(* CODESYS project shelf.library
   Title: Shelf
   Company: Stefan Lehmann
   Version: 0.0.1
   Placeholder: Shelf

Project tree, tasks and I/O mapping:
  libraries: Tc2_System, * (Beckhoff Automation GmbH); Tc2_Utilities, * (Beckhoff Automation GmbH); Tc3_Module, * (Beckhoff Automation GmbH)
  classes/
    function block FifoBuffer [ST]: A_Add, A_Get, A_Remove, A_Reset
    function block Part [ST]: FB_init, id
    function block Shelf [ST]: FB_init, getNextFreeSpace, getNextOccupiedSpace, getShelfSpaceByPartId, m, n, storeNextPart, unloadNextPart, unloadPartById
    function block ShelfElement [ST]: column, isOccupied, part, row, store, unload
  interfaces/
    interface IPart: id
    interface IShelf: getNextFreeSpace, getNextOccupiedSpace, getShelfSpaceByPartId, m, n, storeNextPart, unloadNextPart, unloadPartById
    interface IShelfElement: column, isOccupied, part, row, store, unload
  ClassDiagram
  program main [ST]
*)

// classes/FifoBuffer
FUNCTION_BLOCK FifoBuffer
VAR_INPUT
	bOverwrite	: BOOL;
	in 			: IShelfElement;
END_VAR
VAR_OUTPUT
	bOk			: BOOL;
	nCount		: UDINT;
	nLoad		: UDINT;
	out			: IShelfElement;
END_VAR
VAR
	arrBuffer 	: ARRAY[0..MAX_BUFFER_SIZE] OF BYTE; (* Buffer memory used by FB_MemRingBuffer function block *)
	fbBuffer	: FB_MemRingBuffer;
END_VAR
VAR CONSTANT
	MAX_BUFFER_SIZE : UDINT := 1000;
END_VAR

;

ACTION A_Add:
fbBuffer.A_AddTail( pWrite:= ADR( in ),
					cbWrite:= SIZEOF( in ),
					pBuffer:= ADR( arrBuffer ),
					cbBuffer:= SIZEOF( arrBuffer ),
					bOk=> bOk,
					nCount => nCount );


IF NOT bOk THEN (* overflow ? *)
	IF bOverwrite THEN
		fbBuffer.A_RemoveHead(); (* remove one oldest entry *)

		fbBuffer.A_AddTail( bOk => bOk, nCount => nCount );
	END_IF
END_IF



nLoad := (fbBuffer.cbSize * 100) / MAX_BUFFER_SIZE;
END_ACTION

ACTION A_Get:
fbBuffer.A_GetHead( pRead:= ADR( out ),
					cbRead:= SIZEOF( out ),
					pBuffer:= ADR( arrBuffer ),
					cbBuffer:= SIZEOF( arrBuffer ),
					bOk=> bOk,
					nCount => nCount );

nLoad := (fbBuffer.cbSize * 100) / MAX_BUFFER_SIZE;
END_ACTION

ACTION A_Remove:
fbBuffer.A_RemoveHead( 	pRead:= ADR( out ),
						cbRead:= SIZEOF( out ),
						pBuffer:= ADR( arrBuffer ),
						cbBuffer:= SIZEOF( arrBuffer ),
						bOk=> bOk,
						nCount => nCount );

nLoad := (fbBuffer.cbSize * 100) / MAX_BUFFER_SIZE;
END_ACTION

ACTION A_Reset:
MEMSET( ADR( arrBuffer ), 0, SIZEOF( arrBuffer ) ); (* reset (optional) internal buffer *)

fbBuffer.A_Reset( 	bOk=> bOk,
					nCount => nCount );

nLoad := (fbBuffer.cbSize * 100) / MAX_BUFFER_SIZE;
END_ACTION

END_FUNCTION_BLOCK

// interfaces/IShelfElement
INTERFACE IShelfElement EXTENDS __System.IQueryInterface

PROPERTY column : UINT
GET
END_GET
SET
END_SET
END_PROPERTY

PROPERTY isOccupied : BOOL
GET
END_GET
END_PROPERTY

PROPERTY part : IPart
GET
END_GET
END_PROPERTY

PROPERTY row : UINT
GET
END_GET
SET
END_SET
END_PROPERTY

METHOD store : BOOL
VAR_INPUT
	part: IPart;
END_VAR
END_METHOD

METHOD unload : IPart
VAR_INPUT
END_VAR
END_METHOD

END_INTERFACE

// classes/Part
FUNCTION_BLOCK Part IMPLEMENTS IPart
VAR_INPUT
END_VAR
VAR_OUTPUT
END_VAR
VAR
	_id: STRING(23);
END_VAR

//FB_Init is always available implicitly and it is used primarily for initialization.
//The return value is not evaluated. For a specific influence, you can also declare the
//methods explicitly and provide additional code there with the standard initialization
//code. You can evaluate the return value.
METHOD FB_Init: BOOL
VAR_INPUT
    bInitRetains: BOOL; // TRUE: the retain variables are initialized (reset warm / reset cold)
    bInCopyCode: BOOL;  // TRUE: the instance will be copied to the copy code afterward (online change)
	id: String(23);   
END_VAR
THIS^._id := id;
END_METHOD

{warning 'Eigenschaftenimplementierung hinzufügen'}
PROPERTY id : STRING(23)
GET
id := THIS^._id;
END_GET
SET
THIS^._id := id;
END_SET
END_PROPERTY

END_FUNCTION_BLOCK

// interfaces/IPart
INTERFACE IPart EXTENDS __SYSTEM.IQueryInterface

PROPERTY id : String(23)
GET
END_GET
END_PROPERTY

END_INTERFACE

// classes/Shelf
FUNCTION_BLOCK Shelf IMPLEMENTS IShelf
VAR_INPUT
END_VAR
VAR_OUTPUT
END_VAR
VAR
	rowCount : UINT;
   	columnCount : UINT;
	spaces: ARRAY[0..MAX_ROWS, 0..MAX_COLUMNS] OF ShelfElement();
	freeSpaces: FifoBuffer;
	occupiedSpaces: FifoBuffer;
END_VAR
VAR CONSTANT
	MAX_COLUMNS: INT := 1000;
	MAX_ROWS: INT := 1000;
END_VAR

//FB_Init is always available implicitly and it is used primarily for initialization.
//The return value is not evaluated. For a specific influence, you can also declare the
//methods explicitly and provide additional code there with the standard initialization
//code. You can evaluate the return value.
METHOD FB_Init: BOOL
VAR_INPUT
    bInitRetains: BOOL; // TRUE: the retain variables are initialized (reset warm / reset cold)
    bInCopyCode: BOOL;  // TRUE: the instance will be copied to the copy code afterward (online change)   
	nRows: UINT := 10;
	mColumns: UINT := 10;
END_VAR
VAR
	i: UINT;
	j: UINT;
	k: UINT := 0;
	shelfElement: IShelfElement;
END_VAR
THIS^.rowCount := nRows;
THIS^.columnCount := mColumns;

FOR i:=0 TO nRows - 1 DO
	FOR j:=0 TO mColumns - 1 DO
		shelfElement := THIS^.spaces[i, j];
		shelfElement.row := i;
		shelfElement.column := j;
		THIS^.freeSpaces.A_Add(in := shelfElement); 
	END_FOR
END_FOR
END_METHOD

{warning 'Methodenimplementierung hinzufügen'}
METHOD getNextFreeSpace : IShelfElement
VAR
	freeShelfElement: IShelfElement;
END_VAR
THIS^.freeSpaces.A_Get( out => freeShelfElement);
getNextFreeSpace := freeShelfElement;
END_METHOD

{warning 'Methodenimplementierung hinzufügen'}
METHOD getNextOccupiedSpace : IShelfElement
VAR
	occupiedShelfElement: IShelfElement;
END_VAR
THIS^.occupiedSpaces.A_Get( out => occupiedShelfElement);
getNextOccupiedSpace := occupiedShelfElement;
END_METHOD

{warning 'Methodenimplementierung hinzufügen'}
METHOD getShelfSpaceByPartId : IShelfElement
VAR_INPUT
	partId: String(23);
END_VAR
VAR
	i: UINT;
	j: UINT;
	shelfElement: IShelfElement;
END_VAR
FOR i:=0 TO THIS^.rowCount - 1 DO
	FOR j:=0 TO THIS^.columnCount - 1 DO
		shelfElement := THIS^.spaces[i, j];
		IF NOT(shelfElement.part = 0) THEN
			IF shelfElement.part.id = partId THEN
				getShelfSpaceByPartId := shelfElement;
				RETURN;
			END_IF;
		END_IF
	END_FOR
END_FOR
END_METHOD

{warning 'Add property implementation'}
PROPERTY m : UINT
GET
m := THIS^.columnCount;
END_GET
END_PROPERTY

{warning 'Add property implementation'}
PROPERTY n : UINT
GET
n := THIS^.rowCount;
END_GET
END_PROPERTY

METHOD storeNextPart : BOOL
VAR_INPUT
	part: IPart;
END_VAR
VAR
	shelfElement: IShelfElement;
END_VAR
THIS^.freeSpaces.A_Remove(out=>shelfElement);
IF NOT (shelfElement = 0) THEN
	shelfElement.store(part);
	THIS^.occupiedSpaces.A_Add(in:=shelfElement);
END_IF
END_METHOD

{warning 'Methodenimplementierung hinzufügen'}
METHOD unloadNextPart : IPart
VAR
	shelfElement: IShelfElement;
END_VAR
shelfElement := THIS^.getNextOccupiedSpace();
unloadNextPart := shelfElement.part;
END_METHOD

{warning 'Methodenimplementierung hinzufügen'}
METHOD unloadPartById : IPart
VAR_INPUT
	partId: STRING(23);
END_VAR
VAR
	shelfElement: IShelfElement;
	part: IPart;
END_VAR
shelfElement := THIS^.getShelfSpaceByPartId(partId);
IF NOT(shelfElement = 0) THEN
	unloadPartById := shelfElement.unload();
END_IF
END_METHOD

END_FUNCTION_BLOCK

// interfaces/IShelf
INTERFACE IShelf EXTENDS __SYSTEM.IQueryInterface

METHOD getNextFreeSpace : IShelfElement
VAR_INPUT
END_VAR
END_METHOD

METHOD getNextOccupiedSpace : IShelfElement
VAR_INPUT
END_VAR
END_METHOD

METHOD getShelfSpaceByPartId : IShelfElement
VAR_INPUT
	partId: STRING(23);
END_VAR
END_METHOD

PROPERTY m : UINT
GET
END_GET
END_PROPERTY

PROPERTY n : UINT
GET
END_GET
END_PROPERTY

METHOD storeNextPart : BOOL
VAR_INPUT
	part: IPart;
END_VAR
END_METHOD

METHOD unloadNextPart : IPart
VAR_INPUT
END_VAR
END_METHOD

METHOD unloadPartById : IPart
VAR_INPUT
	partId: STRING(23);
END_VAR
END_METHOD

END_INTERFACE

// classes/ShelfElement
FUNCTION_BLOCK ShelfElement IMPLEMENTS IShelfElement
VAR_INPUT
END_VAR
VAR_OUTPUT
END_VAR
VAR
	_column: UINT;
	_row: UINT;
	_part: IPart;
	_isOccupied: BOOL := FALSE;
END_VAR
VAR CONSTANT
	ID_SIZE: INT := 23;
END_VAR

{warning 'Add property implementation'}
PROPERTY column : UINT
GET
column := THIS^._column;
END_GET
SET
THIS^._column := column;
END_SET
END_PROPERTY

{warning 'Add property implementation'}
PROPERTY isOccupied : BOOL
GET
isOccupied := THIS^._isOccupied;
END_GET
END_PROPERTY

PROPERTY part : IPart
GET
part := THIS^._part;
END_GET
END_PROPERTY

{warning 'Add property implementation'}
PROPERTY row : UINT
GET
row := THIS^._row;
END_GET
SET
THIS^._row := row;
END_SET
END_PROPERTY

METHOD store : BOOL
VAR_INPUT
	part: IPart;
END_VAR
THIS^._part := part;
THIS^._isOccupied := TRUE;
END_METHOD

METHOD unload : IPart
VAR_INPUT
END_VAR
unload := THIS^.part;
THIS^._part := 0;
END_METHOD

END_FUNCTION_BLOCK

// main
PROGRAM main
VAR
	addPart1: BOOL := FALSE;
	addPart2: BOOL := FALSE;
	getShelfSpaceByPartId: BOOL := FALSE;
	shelf: Shelf(2, 2);
	part1: Part('part1');
	part2: Part('part2');
	shelfElement: IShelfElement;
END_VAR

// Main function for testing some functionality

IF addPart1 THEN
	shelf.storeNextPart(part1);
	addPart1 := FALSE;
END_IF;

IF addPart2 THEN
	shelf.storeNextPart(part2);
	addPart2 := FALSE;
END_IF;

IF getShelfSpaceByPartId THEN
	shelfElement := shelf.getShelfSpaceByPartId('part2');
	getShelfSpaceByPartId := FALSE;
END_IF;

END_PROGRAM
